FUNCTION_BLOCK EQUIP_EntryConveyor (* Composite Function Block Type *)
  (* Standard: 61499-2 *)
  (* Version 0.0, 07/01/2026, Schneider Electric, template *)
  PACKAGE Main;
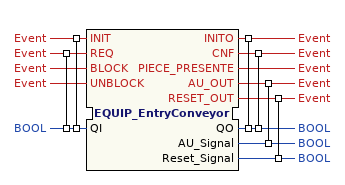
  EVENT_INPUT
    INIT WITH QI; (* Initialization Request *)
    REQ WITH QI; (* Normal Execution Request *)
    BLOCK; (* Bloquer le convoyeur *)
    UNBLOCK; (* Débloquer le convoyeur *)
  END_EVENT
  EVENT_OUTPUT
    INITO WITH QO; (* Initialization Confirm *)
    CNF WITH QO; (* Execution Confirmation *)
    PIECE_PRESENTE;
    AU_OUT WITH AU_Signal; (* Arret urgence active *)
    RESET_OUT WITH Reset_Signal; (* Reset demande *)
  END_EVENT
  VAR_INPUT
    QI : BOOL; (* Input event qualifier *)
  END_VAR
  VAR_OUTPUT
    QO : BOOL; (* Output event qualifier *)
    AU_Signal : BOOL; (* Signal AU pour autres blocs *)
    Reset_Signal : BOOL; (* Signal Reset pour autres blocs *)
  END_VAR
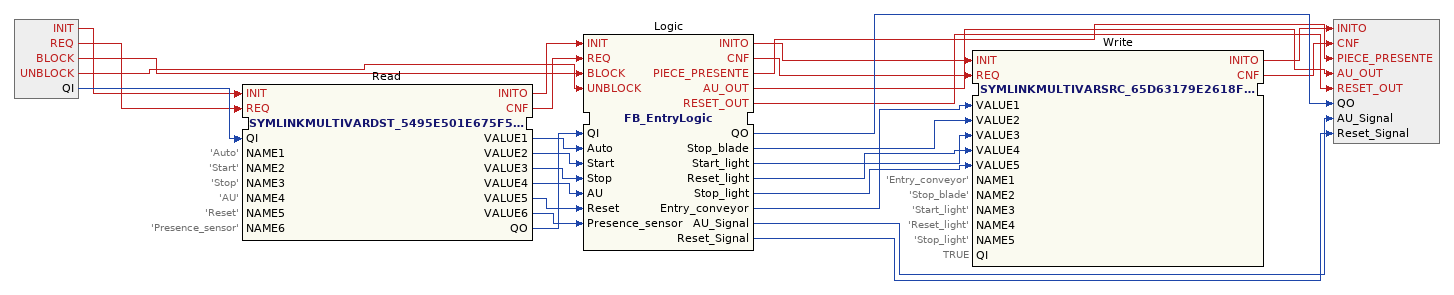
  FBS
    Logic : FB_EntryLogic;
    Write : SYMLINKMULTIVARSRC_65D63179E2618F5E(NAME1 := 'Entry_conveyor', NAME2 := 'Stop_blade', NAME3 := 'Start_light', NAME4 := 'Reset_light', NAME5 := 'Stop_light', QI := TRUE); {SET_ATTRIBUTE(Configuration.GenericFBType.InterfaceParams, Runtime.System#I:=5;VALUE${I$}:BOOL,BOOL,BOOL,BOOL,BOOL)}
    Read : SYMLINKMULTIVARDST_5495E501E675F500(NAME1 := 'Auto', NAME2 := 'Start', NAME3 := 'Stop', NAME4 := 'AU', NAME5 := 'Reset', NAME6 := 'Presence_sensor'); {SET_ATTRIBUTE(Configuration.GenericFBType.InterfaceParams, Runtime.System#I:=6;VALUE${I$}:BOOL,BOOL,BOOL,BOOL,BOOL,BOOL)}
  END_FBS
  EVENT_CONNECTIONS
    INIT TO Read.INIT;
    Read.INITO TO Logic.INIT;
    Logic.INITO TO Write.INIT;
    Write.INITO TO INITO;
    REQ TO Read.REQ;
    Write.CNF TO CNF;
    Read.CNF TO Logic.REQ;
    Logic.CNF TO Write.REQ;
    Logic.PIECE_PRESENTE TO PIECE_PRESENTE;
    BLOCK TO Logic.BLOCK;
    UNBLOCK TO Logic.UNBLOCK;
    Logic.AU_OUT TO AU_OUT;
    Logic.RESET_OUT TO RESET_OUT;
  END_CONNECTIONS
  DATA_CONNECTIONS
    Read.VALUE1 TO Logic.Auto;
    Read.VALUE2 TO Logic.Start;
    Read.VALUE3 TO Logic.Stop;
    Read.VALUE4 TO Logic.AU;
    Read.VALUE5 TO Logic.Reset;
    Read.VALUE6 TO Logic.Presence_sensor;
    Logic.Entry_conveyor TO Write.VALUE1;
    Logic.Stop_blade TO Write.VALUE2;
    Logic.Start_light TO Write.VALUE3;
    Logic.Reset_light TO Write.VALUE4;
    Logic.Stop_light TO Write.VALUE5;
    QI TO Read.QI;
    Logic.QO TO QO;
    Read.QO TO Logic.QI;
    Logic.AU_Signal TO AU_Signal;
    Logic.Reset_Signal TO Reset_Signal;
  END_CONNECTIONS
END_FUNCTION_BLOCK
